LIN {X 0,Y 210.805,Z 412.053,A -85,B 0,C 180,E1 21926.273,E2 21926.273} C_VEL
LIN {X 0,Y 212.909,Z 406.81,A -85,B 0,C 180,E1 21927.449,E2 21927.449} C_VEL
LIN {X 0,Y 212.66,Z 395.692,A -85,B 0,C 180,E1 21932.561,E2 21932.561} C_VEL
LIN {X 0,Y 211.519,Z 388.072,A -85,B 0,C 180,E1 21938.035,E2 21938.035} C_VEL
LIN {X 0,Y 210.505,Z 384.471,A -85,B 0,C 180,E1 21943.363,E2 21943.363} C_VEL
LIN {X 0,Y 210.14,Z 383.897,A -85,B 0,C 180,E1 21947.585,E2 21947.585} C_VEL
LIN {X 0,Y 209.969,Z 386.924,A -85,B 0,C 180,E1 21953.986,E2 21953.986} C_VEL
LIN {X 0,Y 208.207,Z 395.855,A -85,B 0,C 180,E1 21960.026,E2 21960.026} C_VEL
LIN {X 0,Y 204.207,Z 408.112,A -85,B 0,C 180,E1 21965.858,E2 21965.858} C_VEL
LIN {X 0,Y 200.27,Z 414.736,A -85,B 0,C 180,E1 21968.169,E2 21968.169} C_VEL
LIN {X 0,Y 185.94,Z 431.439,A -85,B 0,C 180,E1 21974.122,E2 21974.122} C_VEL
LIN {X 0,Y 172.082,Z 443.956,A -85,B 0,C 180,E1 21982.208,E2 21982.208} C_VEL
LIN {X 0,Y 163.911,Z 449.524,A -85,B 0,C 180,E1 21989.305,E2 21989.305} C_VEL
LIN {X 0,Y 156.576,Z 451.973,A -85,B 0,C 180,E1 21999.559,E2 21999.559} C_VEL
LIN {X 0,Y 153.707,Z 449.459,A -85,B 0,C 180,E1 22009.428,E2 22009.428} C_VEL
LIN {X 0,Y 154.711,Z 442.064,A -85,B 0,C 180,E1 22019.51,E2 22019.51} C_VEL
LIN {X 0,Y 159.246,Z 429.175,A -85,B 0,C 180,E1 22029.201,E2 22029.201} C_VEL
LIN {X 0,Y 161.451,Z 424.273,A -85,B 0,C 180,E1 22032.224,E2 22032.224} C_VEL
LIN {X 0,Y 161.721,Z 426.86,A -85,B 0,C 180,E1 22033.746,E2 22033.746} C_VEL
LIN {X 0,Y 156.787,Z 439.27,A -85,B 0,C 180,E1 22041.701,E2 22041.701} C_VEL
LIN {X 0,Y 154.215,Z 446.583,A -85,B 0,C 180,E1 22050.002,E2 22050.002} C_VEL
LIN {X 0,Y 153.937,Z 447.484,A -85,B 0,C 180,E1 22051.727,E2 22051.727} C_VEL
LIN {X 0,Y 152.482,Z 449.035,A -85,B 0,C 180,E1 22054.89,E2 22054.89} C_VEL
LIN {X 0,Y 147.319,Z 450.78,A -85,B 0,C 180,E1 22063.882,E2 22063.882} C_VEL
LIN {X 0,Y 147.519,Z 450.447,A -85,B 0,C 180,E1 22064.726,E2 22064.726} C_VEL
LIN {X 0,Y 152.99,Z 446.068,A -85,B 0,C 180,E1 22074.785,E2 22074.785} C_VEL
LIN {X 0,Y 160.55,Z 436.902,A -85,B 0,C 180,E1 22083.051,E2 22083.051} C_VEL
LIN {X 0,Y 170.435,Z 421.674,A -85,B 0,C 180,E1 22090.476,E2 22090.476} C_VEL
LIN {X 0,Y 179.907,Z 402.515,A -85,B 0,C 180,E1 22095.907,E2 22095.907} C_VEL
LIN {X 0,Y 183.046,Z 393.253,A -85,B 0,C 180,E1 22097.899,E2 22097.899} C_VEL
LIN {X 0,Y 182.083,Z 375.139,A -85,B 0,C 180,E1 22103.032,E2 22103.032} C_VEL
LIN {X 0,Y 176.944,Z 356.373,A -85,B 0,C 180,E1 22108.755,E2 22108.755} C_VEL
LIN {X 0,Y 167.699,Z 337.888,A -85,B 0,C 180,E1 22116.078,E2 22116.078} C_VEL
LIN {X 0,Y 160.228,Z 325.849,A -85,B 0,C 180,E1 22123.781,E2 22123.781} C_VEL
LIN {X 0,Y 156.957,Z 319.955,A -85,B 0,C 180,E1 22128.879,E2 22128.879} C_VEL
LIN {X 0,Y 154.212,Z 314.241,A -85,B 0,C 180,E1 22136.459,E2 22136.459} C_VEL
LIN {X 0,Y 153.58,Z 313.235,A -85,B 0,C 180,E1 22142.781,E2 22142.781} C_VEL
LIN {X 0,Y 153.957,Z 314.585,A -85,B 0,C 180,E1 22147.024,E2 22147.024} C_VEL
LIN {X 0,Y 157.157,Z 320.346,A -85,B 0,C 180,E1 22155.852,E2 22155.852} C_VEL
LIN {X 0,Y 162.527,Z 330.048,A -85,B 0,C 180,E1 22163.386,E2 22163.386} C_VEL
LIN {X 0,Y 165.204,Z 338.961,A -85,B 0,C 180,E1 22166.589,E2 22166.589} C_VEL
LIN {X 0,Y 174.465,Z 373.972,A -85,B 0,C 180,E1 22175.303,E2 22175.303} C_VEL
LIN {X 0,Y 178.359,Z 393.841,A -85,B 0,C 180,E1 22179.484,E2 22179.484} C_VEL
LIN {X 0,Y 172.426,Z 418.787,A -85,B 0,C 180,E1 22182.402,E2 22182.402} C_VEL
LIN {X 0,Y 164.02,Z 441.927,A -85,B 0,C 180,E1 22187.123,E2 22187.123} C_VEL
LIN {X 0,Y 154.765,Z 462.181,A -85,B 0,C 180,E1 22194.194,E2 22194.194} C_VEL
LIN {X 0,Y 147.761,Z 476.495,A -85,B 0,C 180,E1 22202.64,E2 22202.64} C_VEL
LIN {X 0,Y 144.14,Z 485.452,A -85,B 0,C 180,E1 22211.694,E2 22211.694} C_VEL
LIN {X 0,Y 143.622,Z 488.993,A -85,B 0,C 180,E1 22217.868,E2 22217.868} C_VEL
LIN {X 0,Y 144.238,Z 490.637,A -85,B 0,C 180,E1 22223.993,E2 22223.993} C_VEL
LIN {X 0,Y 145.429,Z 490.426,A -85,B 0,C 180,E1 22229.998,E2 22229.998} C_VEL
LIN {X 0,Y 143.527,Z 490.304,A -85,B 0,C 180,E1 22242.137,E2 22242.137} C_VEL
LIN {X 0,Y 146.123,Z 485.431,A -85,B 0,C 180,E1 22254.396,E2 22254.396} C_VEL
LIN {X 0,Y 156.49,Z 474.216,A -85,B 0,C 180,E1 22267.06,E2 22267.06} C_VEL
LIN {X 0,Y 171.683,Z 458.424,A -85,B 0,C 180,E1 22276.477,E2 22276.477} C_VEL
LIN {X 0,Y 189.39,Z 437.637,A -85,B 0,C 180,E1 22283.408,E2 22283.408} C_VEL
LIN {X 0,Y 206.77,Z 412.673,A -85,B 0,C 180,E1 22288.125,E2 22288.125} C_VEL
LIN {X 0,Y 207.79,Z 406.319,A -85,B 0,C 180,E1 22290.626,E2 22290.626} C_VEL
LIN {X 0,Y 207.548,Z 396.618,A -85,B 0,C 180,E1 22296.457,E2 22296.457} C_VEL
LIN {X 0,Y 206.41,Z 391.41,A -85,B 0,C 180,E1 22303.023,E2 22303.023} C_VEL
LIN {X 0,Y 205.982,Z 390.645,A -85,B 0,C 180,E1 22307.331,E2 22307.331} C_VEL
LIN {X 0,Y 205.755,Z 391.801,A -85,B 0,C 180,E1 22311.592,E2 22311.592} C_VEL
LIN {X 0,Y 204.311,Z 397.423,A -85,B 0,C 180,E1 22316.851,E2 22316.851} C_VEL
LIN {X 0,Y 200.617,Z 407.807,A -85,B 0,C 180,E1 22322.722,E2 22322.722} C_VEL
LIN {X 0,Y 196.464,Z 415.576,A -85,B 0,C 180,E1 22326.12,E2 22326.12} C_VEL
LIN {X 0,Y 180.315,Z 433.31,A -85,B 0,C 180,E1 22332.5,E2 22332.5} C_VEL
LIN {X 0,Y 165.873,Z 445.381,A -85,B 0,C 180,E1 22340.582,E2 22340.582} C_VEL
LIN {X 0,Y 155.739,Z 451.419,A -85,B 0,C 180,E1 22349.308,E2 22349.308} C_VEL
LIN {X 0,Y 149.872,Z 453.121,A -85,B 0,C 180,E1 22357.212,E2 22357.212} C_VEL
LIN {X 0,Y 145.881,Z 450.344,A -85,B 0,C 180,E1 22369.442,E2 22369.442} C_VEL
LIN {X 0,Y 147.229,Z 441.856,A -85,B 0,C 180,E1 22380.841,E2 22380.841} C_VEL
LIN {X 0,Y 152.509,Z 427.688,A -85,B 0,C 180,E1 22391.256,E2 22391.256} C_VEL
LIN {X 0,Y 153.233,Z 427.258,A -85,B 0,C 180,E1 22392.085,E2 22392.085} C_VEL
LIN {X 0,Y 153.723,Z 429.514,A -85,B 0,C 180,E1 22393.609,E2 22393.609} C_VEL
LIN {X 0,Y 148.453,Z 442.037,A -85,B 0,C 180,E1 22402.702,E2 22402.702} C_VEL
LIN {X 0,Y 146.003,Z 449.201,A -85,B 0,C 180,E1 22412.964,E2 22412.964} C_VEL
LIN {X 0,Y 146.669,Z 450.944,A -85,B 0,C 180,E1 22421.876,E2 22421.876} C_VEL
LIN {X 0,Y 147.519,Z 450.447,A -85,B 0,C 180,E1 22424.726,E2 22424.726} C_VEL
LIN {X 0,Y 147.291,Z 449.557,A -85,B 0,C 180,E1 22429.824,E2 22429.824} C_VEL
LIN {X 0,Y 147.002,Z 445.958,A -85,B 0,C 180,E1 22437.425,E2 22437.425} C_VEL
LIN {X 0,Y 147.563,Z 445.28,A -85,B 0,C 180,E1 22438.211,E2 22438.211} C_VEL
LIN {X 0,Y 156.859,Z 433.988,A -85,B 0,C 180,E1 22446.962,E2 22446.962} C_VEL
LIN {X 0,Y 167.545,Z 417.022,A -85,B 0,C 180,E1 22454.121,E2 22454.121} C_VEL
LIN {X 0,Y 177.033,Z 396.635,A -85,B 0,C 180,E1 22459.12,E2 22459.12} C_VEL
LIN {X 0,Y 176.786,Z 379.155,A -85,B 0,C 180,E1 22464.405,E2 22464.405} C_VEL
LIN {X 0,Y 172.627,Z 361.262,A -85,B 0,C 180,E1 22470.275,E2 22470.275} C_VEL
LIN {X 0,Y 165.117,Z 344.486,A -85,B 0,C 180,E1 22477.286,E2 22477.286} C_VEL
LIN {X 0,Y 158.266,Z 332.872,A -85,B 0,C 180,E1 22484.958,E2 22484.958} C_VEL
LIN {X 0,Y 155.4,Z 327.402,A -85,B 0,C 180,E1 22489.872,E2 22489.872} C_VEL
LIN {X 0,Y 153.041,Z 321.347,A -85,B 0,C 180,E1 22497.669,E2 22497.669} C_VEL
LIN {X 0,Y 152.844,Z 322,A -85,B 0,C 180,E1 22506.075,E2 22506.075} C_VEL
LIN {X 0,Y 156.45,Z 329.767,A -85,B 0,C 180,E1 22516.569,E2 22516.569} C_VEL
LIN {X 0,Y 160.808,Z 337.775,A -85,B 0,C 180,E1 22522.738,E2 22522.738} C_VEL
LIN {X 0,Y 168.669,Z 370.735,A -85,B 0,C 180,E1 22531.861,E2 22531.861} C_VEL
LIN {X 0,Y 172.888,Z 396.716,A -85,B 0,C 180,E1 22537.69,E2 22537.69} C_VEL
LIN {X 0,Y 166.006,Z 421.766,A -85,B 0,C 180,E1 22540.92,E2 22540.92} C_VEL
LIN {X 0,Y 156.776,Z 444.406,A -85,B 0,C 180,E1 22546.023,E2 22546.023} C_VEL
LIN {X 0,Y 146.889,Z 463.923,A -85,B 0,C 180,E1 22553.634,E2 22553.634} C_VEL
LIN {X 0,Y 139.622,Z 477.386,A -85,B 0,C 180,E1 22562.654,E2 22562.654} C_VEL
LIN {X 0,Y 135.933,Z 486.411,A -85,B 0,C 180,E1 22573.886,E2 22573.886} C_VEL
LIN {X 0,Y 136.423,Z 489.615,A -85,B 0,C 180,E1 22584.182,E2 22584.182} C_VEL
LIN {X 0,Y 137.542,Z 489.303,A -85,B 0,C 180,E1 22589.998,E2 22589.998} C_VEL
LIN {X 0,Y 135.654,Z 489.171,A -85,B 0,C 180,E1 22602.853,E2 22602.853} C_VEL
LIN {X 0,Y 138.762,Z 484.534,A -85,B 0,C 180,E1 22615.782,E2 22615.782} C_VEL
LIN {X 0,Y 150.121,Z 473.656,A -85,B 0,C 180,E1 22628.918,E2 22628.918} C_VEL
LIN {X 0,Y 167.438,Z 457.052,A -85,B 0,C 180,E1 22639.004,E2 22639.004} C_VEL
LIN {X 0,Y 186.696,Z 435.597,A -85,B 0,C 180,E1 22645.939,E2 22645.939} C_VEL
LIN {X 0,Y 202.13,Z 414.122,A -85,B 0,C 180,E1 22650.063,E2 22650.063} C_VEL
LIN {X 0,Y 202.743,Z 404.443,A -85,B 0,C 180,E1 22655.64,E2 22655.64} C_VEL
LIN {X 0,Y 202.276,Z 398.832,A -85,B 0,C 180,E1 22661.292,E2 22661.292} C_VEL
LIN {X 0,Y 201.541,Z 397.217,A -85,B 0,C 180,E1 22667.047,E2 22667.047} C_VEL
LIN {X 0,Y 201.127,Z 398.232,A -85,B 0,C 180,E1 22671.397,E2 22671.397} C_VEL
LIN {X 0,Y 198.994,Z 403.913,A -85,B 0,C 180,E1 22676.767,E2 22676.767} C_VEL
LIN {X 0,Y 194.16,Z 414.133,A -85,B 0,C 180,E1 22682.645,E2 22682.645} C_VEL
LIN {X 0,Y 190.211,Z 419.697,A -85,B 0,C 180,E1 22684.884,E2 22684.884} C_VEL
LIN {X 0,Y 172.815,Z 436.956,A -85,B 0,C 180,E1 22691.686,E2 22691.686} C_VEL
LIN {X 0,Y 159.581,Z 446.936,A -85,B 0,C 180,E1 22698.991,E2 22698.991} C_VEL
LIN {X 0,Y 150.897,Z 451.871,A -85,B 0,C 180,E1 22705.844,E2 22705.844} C_VEL
LIN {X 0,Y 144.368,Z 454.101,A -85,B 0,C 180,E1 22713.263,E2 22713.263} C_VEL
LIN {X 0,Y 139.14,Z 453.339,A -85,B 0,C 180,E1 22723.652,E2 22723.652} C_VEL
LIN {X 0,Y 138.099,Z 447.736,A -85,B 0,C 180,E1 22735.228,E2 22735.228} C_VEL
LIN {X 0,Y 141.88,Z 436.027,A -85,B 0,C 180,E1 22747.02,E2 22747.02} C_VEL
LIN {X 0,Y 144.913,Z 429.972,A -85,B 0,C 180,E1 22751.798,E2 22751.798} C_VEL
LIN {X 0,Y 146.25,Z 430.872,A -85,B 0,C 180,E1 22752.746,E2 22752.746} C_VEL
LIN {X 0,Y 140.701,Z 443.288,A -85,B 0,C 180,E1 22762.297,E2 22762.297} C_VEL
LIN {X 0,Y 138.16,Z 450.352,A -85,B 0,C 180,E1 22773.132,E2 22773.132} C_VEL
LIN {X 0,Y 139.006,Z 452.016,A -85,B 0,C 180,E1 22782.541,E2 22782.541} C_VEL
LIN {X 0,Y 142.983,Z 449.701,A -85,B 0,C 180,E1 22791.679,E2 22791.679} C_VEL
LIN {X 0,Y 147.563,Z 445.28,A -85,B 0,C 180,E1 22798.211,E2 22798.211} C_VEL
LIN {X 0,Y 149.721,Z 439.575,A -85,B 0,C 180,E1 22804.559,E2 22804.559} C_VEL
LIN {X 0,Y 152.089,Z 432.976,A -85,B 0,C 180,E1 22809.758,E2 22809.758} C_VEL
LIN {X 0,Y 152.872,Z 431.795,A -85,B 0,C 180,E1 22810.388,E2 22810.388} C_VEL
LIN {X 0,Y 163.705,Z 414.626,A -85,B 0,C 180,E1 22816.989,E2 22816.989} C_VEL
LIN {X 0,Y 171.296,Z 398.113,A -85,B 0,C 180,E1 22821.011,E2 22821.011} C_VEL
LIN {X 0,Y 171.365,Z 380.746,A -85,B 0,C 180,E1 22826.61,E2 22826.61} C_VEL
LIN {X 0,Y 167.41,Z 363.025,A -85,B 0,C 180,E1 22833.065,E2 22833.065} C_VEL
LIN {X 0,Y 160.467,Z 346.936,A -85,B 0,C 180,E1 22840.83,E2 22840.83} C_VEL
LIN {X 0,Y 154.104,Z 335.035,A -85,B 0,C 180,E1 22850.453,E2 22850.453} C_VEL
LIN {X 0,Y 151.767,Z 328.746,A -85,B 0,C 180,E1 22859.964,E2 22859.964} C_VEL
LIN {X 0,Y 151.796,Z 329.901,A -85,B 0,C 180,E1 22865.67,E2 22865.67} C_VEL
LIN {X 0,Y 154.905,Z 337.215,A -85,B 0,C 180,E1 22875.684,E2 22875.684} C_VEL
LIN {X 0,Y 158.461,Z 344.268,A -85,B 0,C 180,E1 22881.252,E2 22881.252} C_VEL
LIN {X 0,Y 165.451,Z 378.334,A -85,B 0,C 180,E1 22890.84,E2 22890.84} C_VEL
LIN {X 0,Y 167.53,Z 399.638,A -85,B 0,C 180,E1 22895.837,E2 22895.837} C_VEL
LIN {X 0,Y 159.333,Z 425.462,A -85,B 0,C 180,E1 22899.527,E2 22899.527} C_VEL
LIN {X 0,Y 148.853,Z 448.162,A -85,B 0,C 180,E1 22905.324,E2 22905.324} C_VEL
LIN {X 0,Y 138.78,Z 465.913,A -85,B 0,C 180,E1 22913.269,E2 22913.269} C_VEL
LIN {X 0,Y 131.489,Z 478.074,A -85,B 0,C 180,E1 22922.672,E2 22922.672} C_VEL
LIN {X 0,Y 128.162,Z 485.373,A -85,B 0,C 180,E1 22932.879,E2 22932.879} C_VEL
LIN {X 0,Y 128.366,Z 488.45,A -85,B 0,C 180,E1 22943.247,E2 22943.247} C_VEL
LIN {X 0,Y 129.676,Z 488.176,A -85,B 0,C 180,E1 22949.998,E2 22949.998} C_VEL
LIN {X 0,Y 127.83,Z 488.043,A -85,B 0,C 180,E1 22963.654,E2 22963.654} C_VEL
LIN {X 0,Y 131.494,Z 483.615,A -85,B 0,C 180,E1 22977.323,E2 22977.323} C_VEL
LIN {X 0,Y 143.906,Z 473.073,A -85,B 0,C 180,E1 22990.946,E2 22990.946} C_VEL
LIN {X 0,Y 162.302,Z 456.894,A -85,B 0,C 180,E1 23001.136,E2 23001.136} C_VEL
LIN {X 0,Y 180.943,Z 437.582,A -85,B 0,C 180,E1 23007.604,E2 23007.604} C_VEL
LIN {X 0,Y 196.06,Z 418.633,A -85,B 0,C 180,E1 23011.375,E2 23011.375} C_VEL
LIN {X 0,Y 197.333,Z 413.38,A -85,B 0,C 180,E1 23013.946,E2 23013.946} C_VEL
LIN {X 0,Y 197.677,Z 406.978,A -85,B 0,C 180,E1 23019.037,E2 23019.037} C_VEL
LIN {X 0,Y 197.396,Z 404.738,A -85,B 0,C 180,E1 23022.223,E2 23022.223} C_VEL
LIN {X 0,Y 196.826,Z 403.614,A -85,B 0,C 180,E1 23026.731,E2 23026.731} C_VEL
LIN {X 0,Y 196.239,Z 404.454,A -85,B 0,C 180,E1 23031.181,E2 23031.181} C_VEL
LIN {X 0,Y 194.096,Z 408.723,A -85,B 0,C 180,E1 23035.569,E2 23035.569} C_VEL
LIN {X 0,Y 188.715,Z 418.042,A -85,B 0,C 180,E1 23041.394,E2 23041.394} C_VEL
LIN {X 0,Y 184.124,Z 423.609,A -85,B 0,C 180,E1 23043.541,E2 23043.541} C_VEL
LIN {X 0,Y 168.281,Z 438.119,A -85,B 0,C 180,E1 23049.475,E2 23049.475} C_VEL
LIN {X 0,Y 153.567,Z 448.438,A -85,B 0,C 180,E1 23057.182,E2 23057.182} C_VEL
LIN {X 0,Y 143.496,Z 453.5,A -85,B 0,C 180,E1 23064.917,E2 23064.917} C_VEL
LIN {X 0,Y 133.608,Z 455.364,A -85,B 0,C 180,E1 23077.762,E2 23077.762} C_VEL
LIN {X 0,Y 130.093,Z 451.283,A -85,B 0,C 180,E1 23090.894,E2 23090.894} C_VEL
LIN {X 0,Y 132.032,Z 442.347,A -85,B 0,C 180,E1 23102.798,E2 23102.798} C_VEL
LIN {X 0,Y 136.522,Z 432.65,A -85,B 0,C 180,E1 23111.473,E2 23111.473} C_VEL
LIN {X 0,Y 138.032,Z 433.439,A -85,B 0,C 180,E1 23112.506,E2 23112.506} C_VEL
LIN {X 0,Y 132.977,Z 444.536,A -85,B 0,C 180,E1 23121.847,E2 23121.847} C_VEL
LIN {X 0,Y 130.321,Z 451.504,A -85,B 0,C 180,E1 23133.321,E2 23133.321} C_VEL
LIN {X 0,Y 131.334,Z 453.091,A -85,B 0,C 180,E1 23143.287,E2 23143.287} C_VEL
LIN {X 0,Y 135.672,Z 450.7,A -85,B 0,C 180,E1 23152.912,E2 23152.912} C_VEL
LIN {X 0,Y 143.946,Z 442.74,A -85,B 0,C 180,E1 23163.212,E2 23163.212} C_VEL
LIN {X 0,Y 152.872,Z 431.795,A -85,B 0,C 180,E1 23170.388,E2 23170.388} C_VEL
LIN {X 0,Y 156.693,Z 422.244,A -85,B 0,C 180,E1 23175.64,E2 23175.64} C_VEL
LIN {X 0,Y 159.956,Z 412.576,A -85,B 0,C 180,E1 23179.794,E2 23179.794} C_VEL
LIN {X 0,Y 160.772,Z 410.96,A -85,B 0,C 180,E1 23180.247,E2 23180.247} C_VEL
LIN {X 0,Y 165.708,Z 399.848,A -85,B 0,C 180,E1 23182.948,E2 23182.948} C_VEL
LIN {X 0,Y 166.113,Z 382.865,A -85,B 0,C 180,E1 23188.852,E2 23188.852} C_VEL
LIN {X 0,Y 162.778,Z 365.829,A -85,B 0,C 180,E1 23195.684,E2 23195.684} C_VEL
LIN {X 0,Y 157.291,Z 352.144,A -85,B 0,C 180,E1 23203.237,E2 23203.237} C_VEL
LIN {X 0,Y 152.493,Z 342.283,A -85,B 0,C 180,E1 23211.789,E2 23211.789} C_VEL
LIN {X 0,Y 150.797,Z 336.592,A -85,B 0,C 180,E1 23219.964,E2 23219.964} C_VEL
LIN {X 0,Y 150.78,Z 337.933,A -85,B 0,C 180,E1 23225.528,E2 23225.528} C_VEL
LIN {X 0,Y 153.465,Z 344.797,A -85,B 0,C 180,E1 23234.922,E2 23234.922} C_VEL
LIN {X 0,Y 156.314,Z 351.22,A -85,B 0,C 180,E1 23239.895,E2 23239.895} C_VEL
LIN {X 0,Y 161.485,Z 382.794,A -85,B 0,C 180,E1 23249.038,E2 23249.038} C_VEL
LIN {X 0,Y 162.32,Z 402.187,A -85,B 0,C 180,E1 23253.864,E2 23253.864} C_VEL
LIN {X 0,Y 153.779,Z 426.313,A -85,B 0,C 180,E1 23257.493,E2 23257.493} C_VEL
LIN {X 0,Y 142.508,Z 448.71,A -85,B 0,C 180,E1 23263.494,E2 23263.494} C_VEL
LIN {X 0,Y 131.555,Z 466.294,A -85,B 0,C 180,E1 23271.934,E2 23271.934} C_VEL
LIN {X 0,Y 123.393,Z 478.609,A -85,B 0,C 180,E1 23282.701,E2 23282.701} C_VEL
LIN {X 0,Y 120.059,Z 485.795,A -85,B 0,C 180,E1 23295.439,E2 23295.439} C_VEL
LIN {X 0,Y 120.873,Z 487.433,A -85,B 0,C 180,E1 23306.366,E2 23306.366} C_VEL
LIN {X 0,Y 121.317,Z 486.688,A -85,B 0,C 180,E1 23311.908,E2 23311.908} C_VEL
LIN {X 0,Y 120.005,Z 486.912,A -85,B 0,C 180,E1 23324.563,E2 23324.563} C_VEL
LIN {X 0,Y 126.284,Z 481.233,A -85,B 0,C 180,E1 23341.962,E2 23341.962} C_VEL
LIN {X 0,Y 139.924,Z 471.028,A -85,B 0,C 180,E1 23354.504,E2 23354.504} C_VEL
LIN {X 0,Y 160.011,Z 454.469,A -85,B 0,C 180,E1 23364.426,E2 23364.426} C_VEL
LIN {X 0,Y 179.816,Z 434.786,A -85,B 0,C 180,E1 23370.532,E2 23370.532} C_VEL
LIN {X 0,Y 191.147,Z 421.174,A -85,B 0,C 180,E1 23373.152,E2 23373.152} C_VEL
LIN {X 0,Y 192.528,Z 413.608,A -85,B 0,C 180,E1 23378.568,E2 23378.568} C_VEL
LIN {X 0,Y 192.418,Z 411.209,A -85,B 0,C 180,E1 23381.747,E2 23381.747} C_VEL
LIN {X 0,Y 191.854,Z 409.833,A -85,B 0,C 180,E1 23386.38,E2 23386.38} C_VEL
LIN {X 0,Y 191.109,Z 410.493,A -85,B 0,C 180,E1 23390.942,E2 23390.942} C_VEL
LIN {X 0,Y 188.294,Z 414.857,A -85,B 0,C 180,E1 23395.432,E2 23395.432} C_VEL
LIN {X 0,Y 182.741,Z 422.708,A -85,B 0,C 180,E1 23400.502,E2 23400.502} C_VEL
LIN {X 0,Y 164.382,Z 439.097,A -85,B 0,C 180,E1 23406.999,E2 23406.999} C_VEL
LIN {X 0,Y 146.552,Z 450.584,A -85,B 0,C 180,E1 23415.965,E2 23415.965} C_VEL
LIN {X 0,Y 133.074,Z 456.024,A -85,B 0,C 180,E1 23427.02,E2 23427.02} C_VEL
LIN {X 0,Y 126.093,Z 456.508,A -85,B 0,C 180,E1 23436.808,E2 23436.808} C_VEL
LIN {X 0,Y 122.301,Z 452.626,A -85,B 0,C 180,E1 23449.795,E2 23449.795} C_VEL
LIN {X 0,Y 124.386,Z 442.778,A -85,B 0,C 180,E1 23463.664,E2 23463.664} C_VEL
LIN {X 0,Y 127.906,Z 435.011,A -85,B 0,C 180,E1 23470.835,E2 23470.835} C_VEL
LIN {X 0,Y 129.937,Z 436.257,A -85,B 0,C 180,E1 23472.517,E2 23472.517} C_VEL
LIN {X 0,Y 124.598,Z 447.108,A -85,B 0,C 180,E1 23483.046,E2 23483.046} C_VEL
LIN {X 0,Y 122.496,Z 452.653,A -85,B 0,C 180,E1 23493.533,E2 23493.533} C_VEL
LIN {X 0,Y 123.686,Z 454.166,A -85,B 0,C 180,E1 23504.125,E2 23504.125} C_VEL
LIN {X 0,Y 128.447,Z 451.697,A -85,B 0,C 180,E1 23514.281,E2 23514.281} C_VEL
LIN {X 0,Y 137.57,Z 443.46,A -85,B 0,C 180,E1 23525.163,E2 23525.163} C_VEL
LIN {X 0,Y 148.385,Z 430.671,A -85,B 0,C 180,E1 23533.351,E2 23533.351} C_VEL
LIN {X 0,Y 159.898,Z 412.582,A -85,B 0,C 180,E1 23539.819,E2 23539.819} C_VEL
LIN {X 0,Y 160.772,Z 410.96,A -85,B 0,C 180,E1 23540.247,E2 23540.247} C_VEL
LIN {X 0,Y 162.059,Z 405.175,A -85,B 0,C 180,E1 23542.492,E2 23542.492} C_VEL
LIN {X 0,Y 160.978,Z 396.411,A -85,B 0,C 180,E1 23546.913,E2 23546.913} C_VEL
LIN {X 0,Y 160.558,Z 379.637,A -85,B 0,C 180,E1 23553.447,E2 23553.447} C_VEL
LIN {X 0,Y 156.861,Z 363.892,A -85,B 0,C 180,E1 23561.199,E2 23561.199} C_VEL
LIN {X 0,Y 152.459,Z 353.028,A -85,B 0,C 180,E1 23569.366,E2 23569.366} C_VEL
LIN {X 0,Y 150.687,Z 349.088,A -85,B 0,C 180,E1 23573.988,E2 23573.988} C_VEL
LIN {X 0,Y 149.83,Z 344.417,A -85,B 0,C 180,E1 23579.964,E2 23579.964} C_VEL
LIN {X 0,Y 149.754,Z 345.853,A -85,B 0,C 180,E1 23585.203,E2 23585.203} C_VEL
LIN {X 0,Y 152.127,Z 352.59,A -85,B 0,C 180,E1 23594.322,E2 23594.322} C_VEL
LIN {X 0,Y 154.171,Z 357.768,A -85,B 0,C 180,E1 23598.327,E2 23598.327} C_VEL
LIN {X 0,Y 157.398,Z 386.382,A -85,B 0,C 180,E1 23606.92,E2 23606.92} C_VEL
LIN {X 0,Y 157.312,Z 404.479,A -85,B 0,C 180,E1 23611.75,E2 23611.75} C_VEL
LIN {X 0,Y 147.518,Z 429.048,A -85,B 0,C 180,E1 23615.711,E2 23615.711} C_VEL
LIN {X 0,Y 135.243,Z 450.893,A -85,B 0,C 180,E1 23622.148,E2 23622.148} C_VEL
LIN {X 0,Y 123.57,Z 467.694,A -85,B 0,C 180,E1 23631.253,E2 23631.253} C_VEL
LIN {X 0,Y 115.288,Z 479.002,A -85,B 0,C 180,E1 23642.732,E2 23642.732} C_VEL
LIN {X 0,Y 112.271,Z 484.727,A -85,B 0,C 180,E1 23654.404,E2 23654.404} C_VEL
LIN {X 0,Y 112.491,Z 486.26,A -85,B 0,C 180,E1 23662.289,E2 23662.289} C_VEL
LIN {X 0,Y 113.889,Z 485.895,A -85,B 0,C 180,E1 23669.998,E2 23669.998} C_VEL
LIN {X 0,Y 112.238,Z 485.719,A -85,B 0,C 180,E1 23685.596,E2 23685.596} C_VEL
LIN {X 0,Y 119.281,Z 480.544,A -85,B 0,C 180,E1 23703.777,E2 23703.777} C_VEL
LIN {X 0,Y 135.655,Z 469.585,A -85,B 0,C 180,E1 23717.764,E2 23717.764} C_VEL
LIN {X 0,Y 156.889,Z 453.28,A -85,B 0,C 180,E1 23727.306,E2 23727.306} C_VEL
LIN {X 0,Y 179.167,Z 431.933,A -85,B 0,C 180,E1 23733.489,E2 23733.489} C_VEL
LIN {X 0,Y 185.462,Z 424.819,A -85,B 0,C 180,E1 23734.819,E2 23734.819} C_VEL
LIN {X 0,Y 186.889,Z 420.362,A -85,B 0,C 180,E1 23737.888,E2 23737.888} C_VEL
LIN {X 0,Y 187.131,Z 417.51,A -85,B 0,C 180,E1 23741.212,E2 23741.212} C_VEL
LIN {X 0,Y 186.605,Z 415.856,A -85,B 0,C 180,E1 23746.017,E2 23746.017} C_VEL
LIN {X 0,Y 185.698,Z 416.347,A -85,B 0,C 180,E1 23750.676,E2 23750.676} C_VEL
LIN {X 0,Y 181.541,Z 421.568,A -85,B 0,C 180,E1 23755.892,E2 23755.892} C_VEL
LIN {X 0,Y 177.832,Z 425.976,A -85,B 0,C 180,E1 23758.814,E2 23758.814} C_VEL
LIN {X 0,Y 157.972,Z 442.127,A -85,B 0,C 180,E1 23765.516,E2 23765.516} C_VEL
LIN {X 0,Y 140.138,Z 452.46,A -85,B 0,C 180,E1 23774.284,E2 23774.284} C_VEL
LIN {X 0,Y 129.968,Z 456.39,A -85,B 0,C 180,E1 23781.75,E2 23781.75} C_VEL
LIN {X 0,Y 122.156,Z 457.854,A -85,B 0,C 180,E1 23790.154,E2 23790.154} C_VEL
LIN {X 0,Y 115.289,Z 455.59,A -85,B 0,C 180,E1 23804.342,E2 23804.342} C_VEL
LIN {X 0,Y 114.969,Z 448.327,A -85,B 0,C 180,E1 23818.334,E2 23818.334} C_VEL
LIN {X 0,Y 119.593,Z 437.622,A -85,B 0,C 180,E1 23830.482,E2 23830.482} C_VEL
LIN {X 0,Y 121.648,Z 439.376,A -85,B 0,C 180,E1 23832.902,E2 23832.902} C_VEL
LIN {X 0,Y 116.258,Z 449.535,A -85,B 0,C 180,E1 23844.416,E2 23844.416} C_VEL
LIN {X 0,Y 114.654,Z 454.745,A -85,B 0,C 180,E1 23857.565,E2 23857.565} C_VEL
LIN {X 0,Y 116.069,Z 455.241,A -85,B 0,C 180,E1 23865.073,E2 23865.073} C_VEL
LIN {X 0,Y 121.287,Z 452.698,A -85,B 0,C 180,E1 23875.816,E2 23875.816} C_VEL
LIN {X 0,Y 131.184,Z 444.352,A -85,B 0,C 180,E1 23887.152,E2 23887.152} C_VEL
LIN {X 0,Y 142.732,Z 431.433,A -85,B 0,C 180,E1 23895.533,E2 23895.533} C_VEL
LIN {X 0,Y 154.947,Z 413.14,A -85,B 0,C 180,E1 23902.064,E2 23902.064} C_VEL
LIN {X 0,Y 160.269,Z 401.818,A -85,B 0,C 180,E1 23904.94,E2 23904.94} C_VEL
LIN {X 0,Y 160.978,Z 396.411,A -85,B 0,C 180,E1 23906.913,E2 23906.913} C_VEL
LIN {X 0,Y 159.626,Z 389.093,A -85,B 0,C 180,E1 23910.776,E2 23910.776} C_VEL
LIN {X 0,Y 155.49,Z 378.673,A -85,B 0,C 180,E1 23917.838,E2 23917.838} C_VEL
LIN {X 0,Y 152.589,Z 365.981,A -85,B 0,C 180,E1 23925.466,E2 23925.466} C_VEL
LIN {X 0,Y 149.683,Z 357.153,A -85,B 0,C 180,E1 23933.815,E2 23933.815} C_VEL
LIN {X 0,Y 148.755,Z 352.334,A -85,B 0,C 180,E1 23941.417,E2 23941.417} C_VEL
LIN {X 0,Y 148.808,Z 355.001,A -85,B 0,C 180,E1 23946.332,E2 23946.332} C_VEL
LIN {X 0,Y 150.809,Z 360.325,A -85,B 0,C 180,E1 23953.711,E2 23953.711} C_VEL
LIN {X 0,Y 152.128,Z 364.314,A -85,B 0,C 180,E1 23956.718,E2 23956.718} C_VEL
LIN {X 0,Y 153.43,Z 390.946,A -85,B 0,C 180,E1 23965.06,E2 23965.06} C_VEL
LIN {X 0,Y 152.653,Z 406.086,A -85,B 0,C 180,E1 23969.424,E2 23969.424} C_VEL
LIN {X 0,Y 142.319,Z 429.75,A -85,B 0,C 180,E1 23973.383,E2 23973.383} C_VEL
LIN {X 0,Y 129.981,Z 450.139,A -85,B 0,C 180,E1 23979.518,E2 23979.518} C_VEL
LIN {X 0,Y 117.353,Z 466.806,A -85,B 0,C 180,E1 23988.773,E2 23988.773} C_VEL
LIN {X 0,Y 108.126,Z 478.001,A -85,B 0,C 180,E1 24000.758,E2 24000.758} C_VEL
LIN {X 0,Y 104.507,Z 483.656,A -85,B 0,C 180,E1 24013.212,E2 24013.212} C_VEL
LIN {X 0,Y 104.554,Z 485.162,A -85,B 0,C 180,E1 24021.699,E2 24021.699} C_VEL
LIN {X 0,Y 105.974,Z 484.758,A -85,B 0,C 180,E1 24029.998,E2 24029.998} C_VEL
LIN {X 0,Y 104.5,Z 484.512,A -85,B 0,C 180,E1 24046.784,E2 24046.784} C_VEL
LIN {X 0,Y 110.446,Z 480.927,A -85,B 0,C 180,E1 24063.125,E2 24063.125} C_VEL
LIN {X 0,Y 126.155,Z 471.758,A -85,B 0,C 180,E1 24077.855,E2 24077.855} C_VEL
LIN {X 0,Y 148.416,Z 456.636,A -85,B 0,C 180,E1 24088.374,E2 24088.374} C_VEL
LIN {X 0,Y 171.01,Z 437.373,A -85,B 0,C 180,E1 24094.748,E2 24094.748} C_VEL
LIN {X 0,Y 180.634,Z 427.453,A -85,B 0,C 180,E1 24096.766,E2 24096.766} C_VEL
LIN {X 0,Y 181.503,Z 423.664,A -85,B 0,C 180,E1 24100.607,E2 24100.607} C_VEL
LIN {X 0,Y 181.089,Z 421.688,A -85,B 0,C 180,E1 24105.554,E2 24105.554} C_VEL
LIN {X 0,Y 180.038,Z 421.976,A -85,B 0,C 180,E1 24110.38,E2 24110.38} C_VEL
LIN {X 0,Y 175.68,Z 426.509,A -85,B 0,C 180,E1 24115.103,E2 24115.103} C_VEL
LIN {X 0,Y 171.277,Z 430.697,A -85,B 0,C 180,E1 24117.538,E2 24117.538} C_VEL
LIN {X 0,Y 151.274,Z 445.268,A -85,B 0,C 180,E1 24124.057,E2 24124.057} C_VEL
LIN {X 0,Y 132.623,Z 454.754,A -85,B 0,C 180,E1 24133.196,E2 24133.196} C_VEL
LIN {X 0,Y 117.336,Z 458.941,A -85,B 0,C 180,E1 24145.816,E2 24145.816} C_VEL
LIN {X 0,Y 108.422,Z 457.454,A -85,B 0,C 180,E1 24160.729,E2 24160.729} C_VEL
LIN {X 0,Y 106.689,Z 451.076,A -85,B 0,C 180,E1 24175.548,E2 24175.548} C_VEL
LIN {X 0,Y 110.946,Z 439.866,A -85,B 0,C 180,E1 24189.622,E2 24189.622} C_VEL
LIN {X 0,Y 113.531,Z 441.851,A -85,B 0,C 180,E1 24192.838,E2 24192.838} C_VEL
LIN {X 0,Y 107.926,Z 451.831,A -85,B 0,C 180,E1 24205.994,E2 24205.994} C_VEL
LIN {X 0,Y 106.91,Z 455.914,A -85,B 0,C 180,E1 24218.529,E2 24218.529} C_VEL
LIN {X 0,Y 108.488,Z 456.317,A -85,B 0,C 180,E1 24226.154,E2 24226.154} C_VEL
LIN {X 0,Y 114.235,Z 453.697,A -85,B 0,C 180,E1 24237.54,E2 24237.54} C_VEL
LIN {X 0,Y 124.973,Z 445.243,A -85,B 0,C 180,E1 24249.342,E2 24249.342} C_VEL
LIN {X 0,Y 137.307,Z 432.189,A -85,B 0,C 180,E1 24257.889,E2 24257.889} C_VEL
LIN {X 0,Y 149.974,Z 414.138,A -85,B 0,C 180,E1 24264.332,E2 24264.332} C_VEL
LIN {X 0,Y 154.856,Z 404.456,A -85,B 0,C 180,E1 24266.85,E2 24266.85} C_VEL
LIN {X 0,Y 156.332,Z 387.632,A -85,B 0,C 180,E1 24273.645,E2 24273.645} C_VEL
LIN {X 0,Y 155.49,Z 378.673,A -85,B 0,C 180,E1 24277.838,E2 24277.838} C_VEL
LIN {X 0,Y 153.28,Z 373.334,A -85,B 0,C 180,E1 24282.195,E2 24282.195} C_VEL
LIN {X 0,Y 148.904,Z 368.422,A -85,B 0,C 180,E1 24290.376,E2 24290.376} C_VEL
LIN {X 0,Y 147.817,Z 363.771,A -85,B 0,C 180,E1 24296.122,E2 24296.122} C_VEL
LIN {X 0,Y 147.713,Z 360.172,A -85,B 0,C 180,E1 24302.159,E2 24302.159} C_VEL
LIN {X 0,Y 149.322,Z 368.019,A -85,B 0,C 180,E1 24313.106,E2 24313.106} C_VEL
LIN {X 0,Y 149.907,Z 371.434,A -85,B 0,C 180,E1 24315.285,E2 24315.285} C_VEL
LIN {X 0,Y 149.22,Z 397.655,A -85,B 0,C 180,E1 24323.821,E2 24323.821} C_VEL
LIN {X 0,Y 147.791,Z 408.695,A -85,B 0,C 180,E1 24327.098,E2 24327.098} C_VEL
LIN {X 0,Y 135.938,Z 432.823,A -85,B 0,C 180,E1 24331.418,E2 24331.418} C_VEL
LIN {X 0,Y 122.131,Z 453.125,A -85,B 0,C 180,E1 24338.283,E2 24338.283} C_VEL
LIN {X 0,Y 108.675,Z 468.88,A -85,B 0,C 180,E1 24348.554,E2 24348.554} C_VEL
LIN {X 0,Y 99.068,Z 479.331,A -85,B 0,C 180,E1 24362.806,E2 24362.806} C_VEL
LIN {X 0,Y 96.793,Z 482.585,A -85,B 0,C 180,E1 24371.83,E2 24371.83} C_VEL
LIN {X 0,Y 96.629,Z 484.06,A -85,B 0,C 180,E1 24381.013,E2 24381.013} C_VEL
LIN {X 0,Y 98.086,Z 483.626,A -85,B 0,C 180,E1 24389.997,E2 24389.997} C_VEL
LIN {X 0,Y 97.289,Z 482.811,A -85,B 0,C 180,E1 24394.445,E2 24394.445} C_VEL
LIN {X 0,Y 97.472,Z 483.009,A -85,B 0,C 180,E1 24411.883,E2 24411.883} C_VEL
LIN {X 0,Y 107.182,Z 478.298,A -85,B 0,C 180,E1 24429.817,E2 24429.817} C_VEL
LIN {X 0,Y 126.214,Z 468.153,A -85,B 0,C 180,E1 24443.678,E2 24443.678} C_VEL
LIN {X 0,Y 150.389,Z 452.198,A -85,B 0,C 180,E1 24452.934,E2 24452.934} C_VEL
LIN {X 0,Y 174.5,Z 431.507,A -85,B 0,C 180,E1 24458.498,E2 24458.498} C_VEL
LIN {X 0,Y 175.645,Z 428.923,A -85,B 0,C 180,E1 24460.909,E2 24460.909} C_VEL
LIN {X 0,Y 175.3,Z 427.308,A -85,B 0,C 180,E1 24465.066,E2 24465.066} C_VEL
LIN {X 0,Y 174.116,Z 427.389,A -85,B 0,C 180,E1 24470.05,E2 24470.05} C_VEL
LIN {X 0,Y 170.441,Z 430.59,A -85,B 0,C 180,E1 24473.678,E2 24473.678} C_VEL
LIN {X 0,Y 166.475,Z 433.94,A -85,B 0,C 180,E1 24475.604,E2 24475.604} C_VEL
LIN {X 0,Y 145.99,Z 447.605,A -85,B 0,C 180,E1 24481.957,E2 24481.957} C_VEL
LIN {X 0,Y 127.154,Z 456.273,A -85,B 0,C 180,E1 24490.761,E2 24490.761} C_VEL
LIN {X 0,Y 110.128,Z 460.237,A -85,B 0,C 180,E1 24504.326,E2 24504.326} C_VEL
LIN {X 0,Y 100.302,Z 457.987,A -85,B 0,C 180,E1 24521.22,E2 24521.22} C_VEL
LIN {X 0,Y 99.341,Z 449.683,A -85,B 0,C 180,E1 24539.228,E2 24539.228} C_VEL
LIN {X 0,Y 102.48,Z 442.264,A -85,B 0,C 180,E1 24548.94,E2 24548.94} C_VEL
LIN {X 0,Y 105.026,Z 444.798,A -85,B 0,C 180,E1 24553.303,E2 24553.303} C_VEL
LIN {X 0,Y 100.119,Z 453.017,A -85,B 0,C 180,E1 24565.681,E2 24565.681} C_VEL
LIN {X 0,Y 99.099,Z 456.97,A -85,B 0,C 180,E1 24578.761,E2 24578.761} C_VEL
LIN {X 0,Y 100.951,Z 457.393,A -85,B 0,C 180,E1 24587.397,E2 24587.397} C_VEL
LIN {X 0,Y 107.291,Z 454.697,A -85,B 0,C 180,E1 24599.492,E2 24599.492} C_VEL
LIN {X 0,Y 118.979,Z 446.132,A -85,B 0,C 180,E1 24611.75,E2 24611.75} C_VEL
LIN {X 0,Y 132.13,Z 432.947,A -85,B 0,C 180,E1 24620.437,E2 24620.437} C_VEL
LIN {X 0,Y 145.776,Z 414.244,A -85,B 0,C 180,E1 24626.995,E2 24626.995} C_VEL
LIN {X 0,Y 149.707,Z 406.674,A -85,B 0,C 180,E1 24629.052,E2 24629.052} C_VEL
LIN {X 0,Y 151.711,Z 391.308,A -85,B 0,C 180,E1 24635.737,E2 24635.737} C_VEL
LIN {X 0,Y 150.756,Z 377.471,A -85,B 0,C 180,E1 24643.237,E2 24643.237} C_VEL
LIN {X 0,Y 148.904,Z 368.422,A -85,B 0,C 180,E1 24650.376,E2 24650.376} C_VEL
LIN {X 0,Y 147.558,Z 368.261,A -85,B 0,C 180,E1 24653.757,E2 24653.757} C_VEL
LIN {X 0,Y 146.037,Z 369.793,A -85,B 0,C 180,E1 24658.952,E2 24658.952} C_VEL
LIN {X 0,Y 146.067,Z 369.443,A -85,B 0,C 180,E1 24659.518,E2 24659.518} C_VEL
LIN {X 0,Y 146.26,Z 368.263,A -85,B 0,C 180,E1 24662.55,E2 24662.55} C_VEL
LIN {X 0,Y 147.425,Z 375.778,A -85,B 0,C 180,E1 24672.714,E2 24672.714} C_VEL
LIN {X 0,Y 145.413,Z 399.277,A -85,B 0,C 180,E1 24680.934,E2 24680.934} C_VEL
LIN {X 0,Y 143.084,Z 411.307,A -85,B 0,C 180,E1 24684.642,E2 24684.642} C_VEL
LIN {X 0,Y 130.492,Z 434.517,A -85,B 0,C 180,E1 24689.008,E2 24689.008} C_VEL
LIN {X 0,Y 115.915,Z 453.949,A -85,B 0,C 180,E1 24695.97,E2 24695.97} C_VEL
LIN {X 0,Y 101.253,Z 469.368,A -85,B 0,C 180,E1 24706.997,E2 24706.997} C_VEL
LIN {X 0,Y 91.91,Z 478.312,A -85,B 0,C 180,E1 24720.489,E2 24720.489} C_VEL
LIN {X 0,Y 89.113,Z 481.511,A -85,B 0,C 180,E1 24730.201,E2 24730.201} C_VEL
LIN {X 0,Y 88.698,Z 482.949,A -85,B 0,C 180,E1 24740.202,E2 24740.202} C_VEL
LIN {X 0,Y 90.166,Z 482.489,A -85,B 0,C 180,E1 24749.997,E2 24749.997} C_VEL
LIN {X 0,Y 89.427,Z 481.383,A -85,B 0,C 180,E1 24754.837,E2 24754.837} C_VEL
LIN {X 0,Y 89.193,Z 482.09,A -85,B 0,C 180,E1 24769.775,E2 24769.775} C_VEL
LIN {X 0,Y 98.843,Z 478.408,A -85,B 0,C 180,E1 24790.323,E2 24790.323} C_VEL
LIN {X 0,Y 119.726,Z 468.746,A -85,B 0,C 180,E1 24805.819,E2 24805.819} C_VEL
LIN {X 0,Y 144.802,Z 453.78,A -85,B 0,C 180,E1 24815.122,E2 24815.122} C_VEL
LIN {X 0,Y 168.194,Z 435.532,A -85,B 0,C 180,E1 24820.321,E2 24820.321} C_VEL
LIN {X 0,Y 169.549,Z 433.892,A -85,B 0,C 180,E1 24821.283,E2 24821.283} C_VEL
LIN {X 0,Y 169.276,Z 432.679,A -85,B 0,C 180,E1 24824.521,E2 24824.521} C_VEL
LIN {X 0,Y 167.911,Z 432.595,A -85,B 0,C 180,E1 24829.678,E2 24829.678} C_VEL
LIN {X 0,Y 165.247,Z 434.568,A -85,B 0,C 180,E1 24832.16,E2 24832.16} C_VEL
LIN {X 0,Y 159.469,Z 438.769,A -85,B 0,C 180,E1 24834.146,E2 24834.146} C_VEL
LIN {X 0,Y 139.972,Z 450.327,A -85,B 0,C 180,E1 24840.039,E2 24840.039} C_VEL
LIN {X 0,Y 119.213,Z 458.609,A -85,B 0,C 180,E1 24849.657,E2 24849.657} C_VEL
LIN {X 0,Y 109.942,Z 460.765,A -85,B 0,C 180,E1 24856.108,E2 24856.108} C_VEL
LIN {X 0,Y 99.247,Z 461.341,A -85,B 0,C 180,E1 24867.2,E2 24867.2} C_VEL
LIN {X 0,Y 91.311,Z 457.082,A -85,B 0,C 180,E1 24885.861,E2 24885.861} C_VEL
LIN {X 0,Y 92.442,Z 447.816,A -85,B 0,C 180,E1 24903.577,E2 24903.577} C_VEL
LIN {X 0,Y 94.242,Z 444.803,A -85,B 0,C 180,E1 24908.531,E2 24908.531} C_VEL
LIN {X 0,Y 96.982,Z 446.169,A -85,B 0,C 180,E1 24911.872,E2 24911.872} C_VEL
LIN {X 0,Y 92.323,Z 454.202,A -85,B 0,C 180,E1 24925.315,E2 24925.315} C_VEL
LIN {X 0,Y 91.336,Z 458.083,A -85,B 0,C 180,E1 24939.512,E2 24939.512} C_VEL
LIN {X 0,Y 93.476,Z 458.466,A -85,B 0,C 180,E1 24948.839,E2 24948.839} C_VEL
LIN {X 0,Y 100.508,Z 455.696,A -85,B 0,C 180,E1 24961.703,E2 24961.703} C_VEL
LIN {X 0,Y 113.231,Z 447.022,A -85,B 0,C 180,E1 24974.402,E2 24974.402} C_VEL
LIN {X 0,Y 128.047,Z 432.812,A -85,B 0,C 180,E1 24983.598,E2 24983.598} C_VEL
LIN {X 0,Y 141.627,Z 414.809,A -85,B 0,C 180,E1 24989.676,E2 24989.676} C_VEL
LIN {X 0,Y 144.636,Z 409.217,A -85,B 0,C 180,E1 24991.269,E2 24991.269} C_VEL
LIN {X 0,Y 147.263,Z 394.815,A -85,B 0,C 180,E1 24998.074,E2 24998.074} C_VEL
LIN {X 0,Y 147.181,Z 381.855,A -85,B 0,C 180,E1 25005.868,E2 25005.868} C_VEL
LIN {X 0,Y 146.193,Z 372.294,A -85,B 0,C 180,E1 25014.781,E2 25014.781} C_VEL
LIN {X 0,Y 146.067,Z 369.443,A -85,B 0,C 180,E1 25019.518,E2 25019.518} C_VEL
LIN {X 0,Y 145.729,Z 370.676,A -85,B 0,C 180,E1 25022.201,E2 25022.201} C_VEL
LIN {X 0,Y 144.271,Z 379.362,A -85,B 0,C 180,E1 25027.312,E2 25027.312} C_VEL
LIN {X 0,Y 144.329,Z 379.768,A -85,B 0,C 180,E1 25027.916,E2 25027.916} C_VEL
LIN {X 0,Y 144.716,Z 383.681,A -85,B 0,C 180,E1 25031.809,E2 25031.809} C_VEL
LIN {X 0,Y 140.114,Z 409.313,A -85,B 0,C 180,E1 25040.862,E2 25040.862} C_VEL
LIN {X 0,Y 137.818,Z 415.341,A -85,B 0,C 180,E1 25042.284,E2 25042.284} C_VEL
LIN {X 0,Y 123.784,Z 438.103,A -85,B 0,C 180,E1 25046.942,E2 25046.942} C_VEL
LIN {X 0,Y 107.742,Z 456.957,A -85,B 0,C 180,E1 25054.627,E2 25054.627} C_VEL
LIN {X 0,Y 92.623,Z 470.862,A -85,B 0,C 180,E1 25066.534,E2 25066.534} C_VEL
LIN {X 0,Y 82.894,Z 479.058,A -85,B 0,C 180,E1 25082.827,E2 25082.827} C_VEL
LIN {X 0,Y 80.793,Z 481.833,A -85,B 0,C 180,E1 25099.232,E2 25099.232} C_VEL
LIN {X 0,Y 82.227,Z 481.349,A -85,B 0,C 180,E1 25109.997,E2 25109.997} C_VEL
LIN {X 0,Y 81.242,Z 480.247,A -85,B 0,C 180,E1 25118.005,E2 25118.005} C_VEL
LIN {X 0,Y 85.085,Z 479.976,A -85,B 0,C 180,E1 25142.141,E2 25142.141} C_VEL
LIN {X 0,Y 99.252,Z 475.159,A -85,B 0,C 180,E1 25159.477,E2 25159.477} C_VEL
LIN {X 0,Y 123.395,Z 464.344,A -85,B 0,C 180,E1 25172.445,E2 25172.445} C_VEL
LIN {X 0,Y 150.45,Z 447.929,A -85,B 0,C 180,E1 25180.098,E2 25180.098} C_VEL
LIN {X 0,Y 162.334,Z 438.948,A -85,B 0,C 180,E1 25182.336,E2 25182.336} C_VEL
LIN {X 0,Y 163.045,Z 437.779,A -85,B 0,C 180,E1 25183.914,E2 25183.914} C_VEL
LIN {X 0,Y 161.426,Z 437.577,A -85,B 0,C 180,E1 25189.258,E2 25189.258} C_VEL
LIN {X 0,Y 157.334,Z 440.254,A -85,B 0,C 180,E1 25191.412,E2 25191.412} C_VEL
LIN {X 0,Y 135.954,Z 452.179,A -85,B 0,C 180,E1 25197.319,E2 25197.319} C_VEL
LIN {X 0,Y 112.343,Z 460.554,A -85,B 0,C 180,E1 25207.768,E2 25207.768} C_VEL
LIN {X 0,Y 96.449,Z 462.692,A -85,B 0,C 180,E1 25220.168,E2 25220.168} C_VEL
LIN {X 0,Y 84.781,Z 459.628,A -85,B 0,C 180,E1 25239.79,E2 25239.79} C_VEL
LIN {X 0,Y 83.757,Z 450.863,A -85,B 0,C 180,E1 25260.507,E2 25260.507} C_VEL
LIN {X 0,Y 85.736,Z 447.033,A -85,B 0,C 180,E1 25267.49,E2 25267.49} C_VEL
LIN {X 0,Y 88.953,Z 449.018,A -85,B 0,C 180,E1 25272.733,E2 25272.733} C_VEL
LIN {X 0,Y 83.633,Z 457.111,A -85,B 0,C 180,E1 25290.003,E2 25290.003} C_VEL
LIN {X 0,Y 83.59,Z 459.197,A -85,B 0,C 180,E1 25300.403,E2 25300.403} C_VEL
LIN {X 0,Y 86.062,Z 459.536,A -85,B 0,C 180,E1 25310.532,E2 25310.532} C_VEL
LIN {X 0,Y 93.892,Z 456.69,A -85,B 0,C 180,E1 25324.232,E2 25324.232} C_VEL
LIN {X 0,Y 107.741,Z 447.913,A -85,B 0,C 180,E1 25337.336,E2 25337.336} C_VEL
LIN {X 0,Y 123.511,Z 433.573,A -85,B 0,C 180,E1 25346.557,E2 25346.557} C_VEL
LIN {X 0,Y 137.813,Z 415.364,A -85,B 0,C 180,E1 25352.516,E2 25352.516} C_VEL
LIN {X 0,Y 140.605,Z 409.126,A -85,B 0,C 180,E1 25354.964,E2 25354.964} C_VEL
LIN {X 0,Y 143.286,Z 395.846,A -85,B 0,C 180,E1 25361.989,E2 25361.989} C_VEL
LIN {X 0,Y 143.721,Z 385.004,A -85,B 0,C 180,E1 25369.827,E2 25369.827} C_VEL
LIN {X 0,Y 143.781,Z 378.47,A -85,B 0,C 180,E1 25377.707,E2 25377.707} C_VEL
LIN {X 0,Y 144.325,Z 376.203,A -85,B 0,C 180,E1 25382.397,E2 25382.397} C_VEL
LIN {X 0,Y 144.329,Z 379.768,A -85,B 0,C 180,E1 25387.916,E2 25387.916} C_VEL
LIN {X 0,Y 143.882,Z 383.892,A -85,B 0,C 180,E1 25390.121,E2 25390.121} C_VEL
LIN {X 0,Y 139.642,Z 398.733,A -85,B 0,C 180,E1 25393.333,E2 25393.333} C_VEL
LIN {X 0,Y 134.949,Z 414.997,A -85,B 0,C 180,E1 25399.166,E2 25399.166} C_VEL
LIN {X 0,Y 121.145,Z 436.407,A -85,B 0,C 180,E1 25403.267,E2 25403.267} C_VEL
LIN {X 0,Y 104.738,Z 454.762,A -85,B 0,C 180,E1 25410.177,E2 25410.177} C_VEL
LIN {X 0,Y 89.359,Z 468.062,A -85,B 0,C 180,E1 25420.54,E2 25420.54} C_VEL
LIN {X 0,Y 78.18,Z 476.267,A -85,B 0,C 180,E1 25434.612,E2 25434.612} C_VEL
LIN {X 0,Y 74.076,Z 479.368,A -85,B 0,C 180,E1 25445.954,E2 25445.954} C_VEL
LIN {X 0,Y 72.895,Z 480.713,A -85,B 0,C 180,E1 25458.049,E2 25458.049} C_VEL
LIN {X 0,Y 74.288,Z 480.209,A -85,B 0,C 180,E1 25469.997,E2 25469.997} C_VEL
LIN {X 0,Y 73.425,Z 478.784,A -85,B 0,C 180,E1 25478.863,E2 25478.863} C_VEL
LIN {X 0,Y 78.366,Z 478.854,A -85,B 0,C 180,E1 25505.283,E2 25505.283} C_VEL
LIN {X 0,Y 94.19,Z 474.339,A -85,B 0,C 180,E1 25523.225,E2 25523.225} C_VEL
LIN {X 0,Y 119.888,Z 463.996,A -85,B 0,C 180,E1 25535.853,E2 25535.853} C_VEL
LIN {X 0,Y 147.936,Z 448.172,A -85,B 0,C 180,E1 25542.99,E2 25542.99} C_VEL
LIN {X 0,Y 154.863,Z 443.418,A -85,B 0,C 180,E1 25544.195,E2 25544.195} C_VEL
LIN {X 0,Y 156.041,Z 442.31,A -85,B 0,C 180,E1 25545.245,E2 25545.245} C_VEL
LIN {X 0,Y 153.724,Z 442.897,A -85,B 0,C 180,E1 25548.991,E2 25548.991} C_VEL
LIN {X 0,Y 128.896,Z 455.389,A -85,B 0,C 180,E1 25555.52,E2 25555.52} C_VEL
LIN {X 0,Y 106.088,Z 462.26,A -85,B 0,C 180,E1 25565.353,E2 25565.353} C_VEL
LIN {X 0,Y 87.371,Z 463.77,A -85,B 0,C 180,E1 25580.274,E2 25580.274} C_VEL
LIN {X 0,Y 76.275,Z 459.492,A -85,B 0,C 180,E1 25601.787,E2 25601.787} C_VEL
LIN {X 0,Y 76.512,Z 449.953,A -85,B 0,C 180,E1 25623.872,E2 25623.872} C_VEL
LIN {X 0,Y 77.689,Z 449.508,A -85,B 0,C 180,E1 25627.144,E2 25627.144} C_VEL
LIN {X 0,Y 79.951,Z 450.625,A -85,B 0,C 180,E1 25630.892,E2 25630.892} C_VEL
LIN {X 0,Y 79.69,Z 452.546,A -85,B 0,C 180,E1 25634.998,E2 25634.998} C_VEL
LIN {X 0,Y 75.607,Z 458.817,A -85,B 0,C 180,E1 25652.285,E2 25652.285} C_VEL
LIN {X 0,Y 78.745,Z 460.598,A -85,B 0,C 180,E1 25672.539,E2 25672.539} C_VEL
LIN {X 0,Y 87.494,Z 457.676,A -85,B 0,C 180,E1 25687.135,E2 25687.135} C_VEL
LIN {X 0,Y 102.557,Z 448.802,A -85,B 0,C 180,E1 25700.58,E2 25700.58} C_VEL
LIN {X 0,Y 119.09,Z 434.584,A -85,B 0,C 180,E1 25709.607,E2 25709.607} C_VEL
LIN {X 0,Y 134.353,Z 415.934,A -85,B 0,C 180,E1 25715.503,E2 25715.503} C_VEL
LIN {X 0,Y 138.317,Z 404.301,A -85,B 0,C 180,E1 25721.68,E2 25721.68} C_VEL
LIN {X 0,Y 140.298,Z 392.802,A -85,B 0,C 180,E1 25729.808,E2 25729.808} C_VEL
LIN {X 0,Y 141.059,Z 386.568,A -85,B 0,C 180,E1 25736.785,E2 25736.785} C_VEL
LIN {X 0,Y 141.864,Z 383.809,A -85,B 0,C 180,E1 25741.569,E2 25741.569} C_VEL
LIN {X 0,Y 141.815,Z 389.502,A -85,B 0,C 180,E1 25749.919,E2 25749.919} C_VEL
LIN {X 0,Y 139.642,Z 398.733,A -85,B 0,C 180,E1 25753.333,E2 25753.333} C_VEL
LIN {X 0,Y 137.039,Z 406.075,A -85,B 0,C 180,E1 25755.035,E2 25755.035} C_VEL
LIN {X 0,Y 129.965,Z 419.018,A -85,B 0,C 180,E1 25756.531,E2 25756.531} C_VEL
LIN {X 0,Y 114.939,Z 439.63,A -85,B 0,C 180,E1 25760.699,E2 25760.699} C_VEL
LIN {X 0,Y 96.508,Z 457.788,A -85,B 0,C 180,E1 25768.411,E2 25768.411} C_VEL
LIN {X 0,Y 79.544,Z 470.302,A -85,B 0,C 180,E1 25780.635,E2 25780.635} C_VEL
LIN {X 0,Y 68.794,Z 476.97,A -85,B 0,C 180,E1 25796.74,E2 25796.74} C_VEL
LIN {X 0,Y 65.044,Z 479.593,A -85,B 0,C 180,E1 25816.581,E2 25816.581} C_VEL
LIN {X 0,Y 66.329,Z 479.066,A -85,B 0,C 180,E1 25829.996,E2 25829.996} C_VEL
LIN {X 0,Y 65.598,Z 477.295,A -85,B 0,C 180,E1 25839.931,E2 25839.931} C_VEL
LIN {X 0,Y 71.904,Z 477.705,A -85,B 0,C 180,E1 25869.015,E2 25869.015} C_VEL
LIN {X 0,Y 94.721,Z 472.012,A -85,B 0,C 180,E1 25890.432,E2 25890.432} C_VEL
LIN {X 0,Y 123.449,Z 460.665,A -85,B 0,C 180,E1 25901.315,E2 25901.315} C_VEL
LIN {X 0,Y 147.088,Z 447.646,A -85,B 0,C 180,E1 25906.183,E2 25906.183} C_VEL
LIN {X 0,Y 147.614,Z 447.118,A -85,B 0,C 180,E1 25907.01,E2 25907.01} C_VEL
LIN {X 0,Y 121.458,Z 458.589,A -85,B 0,C 180,E1 25913.66,E2 25913.66} C_VEL
LIN {X 0,Y 105.183,Z 463.019,A -85,B 0,C 180,E1 25920.051,E2 25920.051} C_VEL
LIN {X 0,Y 89.047,Z 465.095,A -85,B 0,C 180,E1 25929.818,E2 25929.818} C_VEL
LIN {X 0,Y 76.028,Z 464.175,A -85,B 0,C 180,E1 25943.466,E2 25943.466} C_VEL
LIN {X 0,Y 67.396,Z 457.939,A -85,B 0,C 180,E1 25967.806,E2 25967.806} C_VEL
LIN {X 0,Y 68.489,Z 451.153,A -85,B 0,C 180,E1 25983.858,E2 25983.858} C_VEL
LIN {X 0,Y 71.039,Z 452.553,A -85,B 0,C 180,E1 25989.455,E2 25989.455} C_VEL
LIN {X 0,Y 71.959,Z 453.988,A -85,B 0,C 180,E1 25993.856,E2 25993.856} C_VEL
LIN {X 0,Y 67.924,Z 459.451,A -85,B 0,C 180,E1 26010.004,E2 26010.004} C_VEL
LIN {X 0,Y 68.184,Z 461.422,A -85,B 0,C 180,E1 26022.79,E2 26022.79} C_VEL
LIN {X 0,Y 71.536,Z 461.656,A -85,B 0,C 180,E1 26034.957,E2 26034.957} C_VEL
LIN {X 0,Y 81.34,Z 458.659,A -85,B 0,C 180,E1 26050.493,E2 26050.493} C_VEL
LIN {X 0,Y 97.733,Z 449.688,A -85,B 0,C 180,E1 26064.159,E2 26064.159} C_VEL
LIN {X 0,Y 114.518,Z 436.078,A -85,B 0,C 180,E1 26072.684,E2 26072.684} C_VEL
LIN {X 0,Y 129.982,Z 418.326,A -85,B 0,C 180,E1 26078.244,E2 26078.244} C_VEL
LIN {X 0,Y 134.463,Z 407.21,A -85,B 0,C 180,E1 26084.754,E2 26084.754} C_VEL
LIN {X 0,Y 136.944,Z 397.549,A -85,B 0,C 180,E1 26092.633,E2 26092.633} C_VEL
LIN {X 0,Y 138.479,Z 392.368,A -85,B 0,C 180,E1 26099.961,E2 26099.961} C_VEL
LIN {X 0,Y 138.789,Z 392.279,A -85,B 0,C 180,E1 26103.247,E2 26103.247} C_VEL
LIN {X 0,Y 138.742,Z 395.09,A -85,B 0,C 180,E1 26107.93,E2 26107.93} C_VEL
LIN {X 0,Y 131.768,Z 415.715,A -85,B 0,C 180,E1 26115.873,E2 26115.873} C_VEL
LIN {X 0,Y 129.965,Z 419.018,A -85,B 0,C 180,E1 26116.531,E2 26116.531} C_VEL
LIN {X 0,Y 122.476,Z 428.271,A -85,B 0,C 180,E1 26116.365,E2 26116.365} C_VEL
LIN {X 0,Y 115.207,Z 435.721,A -85,B 0,C 180,E1 26116.113,E2 26116.113} C_VEL
LIN {X 0,Y 114.261,Z 436.758,A -85,B 0,C 180,E1 26116.321,E2 26116.321} C_VEL
LIN {X 0,Y 95.503,Z 454.857,A -85,B 0,C 180,E1 26122.819,E2 26122.819} C_VEL
LIN {X 0,Y 77.073,Z 467.815,A -85,B 0,C 180,E1 26133.679,E2 26133.679} C_VEL
LIN {X 0,Y 62.181,Z 475.918,A -85,B 0,C 180,E1 26152.644,E2 26152.644} C_VEL
LIN {X 0,Y 57.224,Z 478.471,A -85,B 0,C 180,E1 26174.706,E2 26174.706} C_VEL
LIN {X 0,Y 58.387,Z 477.924,A -85,B 0,C 180,E1 26189.996,E2 26189.996} C_VEL
LIN {X 0,Y 57.778,Z 475.738,A -85,B 0,C 180,E1 26201.292,E2 26201.292} C_VEL
LIN {X 0,Y 65.828,Z 476.478,A -85,B 0,C 180,E1 26233.443,E2 26233.443} C_VEL
LIN {X 0,Y 90.517,Z 471.408,A -85,B 0,C 180,E1 26254.624,E2 26254.624} C_VEL
LIN {X 0,Y 121.122,Z 460.5,A -85,B 0,C 180,E1 26264.905,E2 26264.905} C_VEL
LIN {X 0,Y 128.778,Z 456.961,A -85,B 0,C 180,E1 26266.489,E2 26266.489} C_VEL
LIN {X 0,Y 129.391,Z 456.47,A -85,B 0,C 180,E1 26267.402,E2 26267.402} C_VEL
LIN {X 0,Y 106.145,Z 463.496,A -85,B 0,C 180,E1 26274.326,E2 26274.326} C_VEL
LIN {X 0,Y 90.572,Z 465.957,A -85,B 0,C 180,E1 26281.633,E2 26281.633} C_VEL
LIN {X 0,Y 76.996,Z 466.191,A -85,B 0,C 180,E1 26291.518,E2 26291.518} C_VEL
LIN {X 0,Y 62.127,Z 462.125,A -85,B 0,C 180,E1 26314.633,E2 26314.633} C_VEL
LIN {X 0,Y 60.436,Z 453.598,A -85,B 0,C 180,E1 26343.072,E2 26343.072} C_VEL
LIN {X 0,Y 63.751,Z 455.27,A -85,B 0,C 180,E1 26351.497,E2 26351.497} C_VEL
LIN {X 0,Y 60.076,Z 460.615,A -85,B 0,C 180,E1 26370.004,E2 26370.004} C_VEL
LIN {X 0,Y 60.537,Z 462.536,A -85,B 0,C 180,E1 26384.438,E2 26384.438} C_VEL
LIN {X 0,Y 64.511,Z 462.709,A -85,B 0,C 180,E1 26397.897,E2 26397.897} C_VEL
LIN {X 0,Y 77.565,Z 458.823,A -85,B 0,C 180,E1 26416.485,E2 26416.485} C_VEL
LIN {X 0,Y 93.321,Z 450.567,A -85,B 0,C 180,E1 26428.1,E2 26428.1} C_VEL
LIN {X 0,Y 112.444,Z 435.619,A -85,B 0,C 180,E1 26436.785,E2 26436.785} C_VEL
LIN {X 0,Y 126.243,Z 420.087,A -85,B 0,C 180,E1 26441.555,E2 26441.555} C_VEL
LIN {X 0,Y 130.947,Z 409.905,A -85,B 0,C 180,E1 26448.323,E2 26448.323} C_VEL
LIN {X 0,Y 133.591,Z 402.815,A -85,B 0,C 180,E1 26455.041,E2 26455.041} C_VEL
LIN {X 0,Y 134.984,Z 399.725,A -85,B 0,C 180,E1 26459.96,E2 26459.96} C_VEL
LIN {X 0,Y 135.268,Z 400.493,A -85,B 0,C 180,E1 26464.847,E2 26464.847} C_VEL
LIN {X 0,Y 134.595,Z 402.865,A -85,B 0,C 180,E1 26466.785,E2 26466.785} C_VEL
LIN {X 0,Y 127.123,Z 419.796,A -85,B 0,C 180,E1 26473.273,E2 26473.273} C_VEL
LIN {X 0,Y 114.261,Z 436.758,A -85,B 0,C 180,E1 26476.321,E2 26476.321} C_VEL
LIN {X 0,Y 101.328,Z 448.297,A -85,B 0,C 180,E1 26477.881,E2 26477.881} C_VEL
LIN {X 0,Y 88.966,Z 456.812,A -85,B 0,C 180,E1 26479.774,E2 26479.774} C_VEL
LIN {X 0,Y 87.345,Z 457.909,A -85,B 0,C 180,E1 26480.393,E2 26480.393} C_VEL
LIN {X 0,Y 67.871,Z 469.486,A -85,B 0,C 180,E1 26492.33,E2 26492.33} C_VEL
LIN {X 0,Y 52.775,Z 476.147,A -85,B 0,C 180,E1 26515.114,E2 26515.114} C_VEL
LIN {X 0,Y 49.494,Z 477.349,A -85,B 0,C 180,E1 26532.244,E2 26532.244} C_VEL
LIN {X 0,Y 50.432,Z 476.775,A -85,B 0,C 180,E1 26549.995,E2 26549.995} C_VEL
LIN {X 0,Y 50.075,Z 474.533,A -85,B 0,C 180,E1 26567.533,E2 26567.533} C_VEL
LIN {X 0,Y 60.215,Z 475.252,A -85,B 0,C 180,E1 26598.74,E2 26598.74} C_VEL
LIN {X 0,Y 82.011,Z 471.874,A -85,B 0,C 180,E1 26616.918,E2 26616.918} C_VEL
LIN {X 0,Y 108.696,Z 464.313,A -85,B 0,C 180,E1 26626.349,E2 26626.349} C_VEL
LIN {X 0,Y 111.504,Z 463.094,A -85,B 0,C 180,E1 26627.849,E2 26627.849} C_VEL
LIN {X 0,Y 90.859,Z 466.866,A -85,B 0,C 180,E1 26635.162,E2 26635.162} C_VEL
LIN {X 0,Y 75.625,Z 467.569,A -85,B 0,C 180,E1 26643.952,E2 26643.952} C_VEL
LIN {X 0,Y 56.987,Z 464.197,A -85,B 0,C 180,E1 26666.341,E2 26666.341} C_VEL
LIN {X 0,Y 52.1,Z 455.664,A -85,B 0,C 180,E1 26700.544,E2 26700.544} C_VEL
LIN {X 0,Y 54.464,Z 456.82,A -85,B 0,C 180,E1 26708.194,E2 26708.194} C_VEL
LIN {X 0,Y 55.347,Z 458.056,A -85,B 0,C 180,E1 26714.183,E2 26714.183} C_VEL
LIN {X 0,Y 52.22,Z 461.774,A -85,B 0,C 180,E1 26730.005,E2 26730.005} C_VEL
LIN {X 0,Y 52.958,Z 463.648,A -85,B 0,C 180,E1 26746.56,E2 26746.56} C_VEL
LIN {X 0,Y 57.669,Z 463.767,A -85,B 0,C 180,E1 26761.561,E2 26761.561} C_VEL
LIN {X 0,Y 72.981,Z 459.565,A -85,B 0,C 180,E1 26781.567,E2 26781.567} C_VEL
LIN {X 0,Y 92.443,Z 449.569,A -85,B 0,C 180,E1 26793.875,E2 26793.875} C_VEL
LIN {X 0,Y 111.569,Z 434.476,A -85,B 0,C 180,E1 26801.228,E2 26801.228} C_VEL
LIN {X 0,Y 122.503,Z 422.438,A -85,B 0,C 180,E1 26804.78,E2 26804.78} C_VEL
LIN {X 0,Y 127.36,Z 413.719,A -85,B 0,C 180,E1 26811.303,E2 26811.303} C_VEL
LIN {X 0,Y 129.834,Z 408.829,A -85,B 0,C 180,E1 26816.627,E2 26816.627} C_VEL
LIN {X 0,Y 131.049,Z 406.905,A -85,B 0,C 180,E1 26819.959,E2 26819.959} C_VEL
LIN {X 0,Y 131.442,Z 407.213,A -85,B 0,C 180,E1 26824.074,E2 26824.074} C_VEL
LIN {X 0,Y 124.546,Z 420.719,A -85,B 0,C 180,E1 26829.871,E2 26829.871} C_VEL
LIN {X 0,Y 106.809,Z 441.769,A -85,B 0,C 180,E1 26833.752,E2 26833.752} C_VEL
LIN {X 0,Y 87.345,Z 457.909,A -85,B 0,C 180,E1 26840.393,E2 26840.393} C_VEL
LIN {X 0,Y 72.6,Z 465.556,A -85,B 0,C 180,E1 26844.515,E2 26844.515} C_VEL
LIN {X 0,Y 59.458,Z 470.429,A -85,B 0,C 180,E1 26850.019,E2 26850.019} C_VEL
LIN {X 0,Y 57.898,Z 471.005,A -85,B 0,C 180,E1 26851.413,E2 26851.413} C_VEL
LIN {X 0,Y 46.35,Z 475.074,A -85,B 0,C 180,E1 26869.366,E2 26869.366} C_VEL
LIN {X 0,Y 41.877,Z 476.226,A -85,B 0,C 180,E1 26888.873,E2 26888.873} C_VEL
LIN {X 0,Y 42.475,Z 475.619,A -85,B 0,C 180,E1 26909.994,E2 26909.994} C_VEL
LIN {X 0,Y 42.554,Z 472.901,A -85,B 0,C 180,E1 26930.763,E2 26930.763} C_VEL
LIN {X 0,Y 59.399,Z 473.709,A -85,B 0,C 180,E1 26969.568,E2 26969.568} C_VEL
LIN {X 0,Y 87.321,Z 469.318,A -85,B 0,C 180,E1 26985.399,E2 26985.399} C_VEL
LIN {X 0,Y 94.216,Z 467.507,A -85,B 0,C 180,E1 26988.198,E2 26988.198} C_VEL
LIN {X 0,Y 69.391,Z 468.645,A -85,B 0,C 180,E1 27000.078,E2 27000.078} C_VEL
LIN {X 0,Y 49.439,Z 464.671,A -85,B 0,C 180,E1 27023.71,E2 27023.71} C_VEL
LIN {X 0,Y 43.689,Z 457.431,A -85,B 0,C 180,E1 27055.138,E2 27055.138} C_VEL
LIN {X 0,Y 47.153,Z 459.374,A -85,B 0,C 180,E1 27071.341,E2 27071.341} C_VEL
LIN {X 0,Y 44.365,Z 462.926,A -85,B 0,C 180,E1 27090.006,E2 27090.006} C_VEL
LIN {X 0,Y 45.491,Z 464.759,A -85,B 0,C 180,E1 27109.379,E2 27109.379} C_VEL
LIN {X 0,Y 51.143,Z 464.821,A -85,B 0,C 180,E1 27126.171,E2 27126.171} C_VEL
LIN {X 0,Y 66.706,Z 461.102,A -85,B 0,C 180,E1 27145.426,E2 27145.426} C_VEL
LIN {X 0,Y 86.019,Z 452.315,A -85,B 0,C 180,E1 27157.078,E2 27157.078} C_VEL
LIN {X 0,Y 106.428,Z 437.786,A -85,B 0,C 180,E1 27164.357,E2 27164.357} C_VEL
LIN {X 0,Y 118.502,Z 425.635,A -85,B 0,C 180,E1 27167.723,E2 27167.723} C_VEL
LIN {X 0,Y 123.757,Z 417.85,A -85,B 0,C 180,E1 27174.306,E2 27174.306} C_VEL
LIN {X 0,Y 126.577,Z 413.883,A -85,B 0,C 180,E1 27179.957,E2 27179.957} C_VEL
LIN {X 0,Y 127.022,Z 413.517,A -85,B 0,C 180,E1 27181.524,E2 27181.524} C_VEL
LIN {X 0,Y 125.75,Z 415.911,A -85,B 0,C 180,E1 27183.559,E2 27183.559} C_VEL
LIN {X 0,Y 120.647,Z 423.979,A -85,B 0,C 180,E1 27186.71,E2 27186.71} C_VEL
LIN {X 0,Y 101.61,Z 444.277,A -85,B 0,C 180,E1 27190.292,E2 27190.292} C_VEL
LIN {X 0,Y 79.131,Z 460.626,A -85,B 0,C 180,E1 27197.534,E2 27197.534} C_VEL
LIN {X 0,Y 57.898,Z 471.005,A -85,B 0,C 180,E1 27211.413,E2 27211.413} C_VEL
LIN {X 0,Y 44.479,Z 474.341,A -85,B 0,C 180,E1 27223.621,E2 27223.621} C_VEL
LIN {X 0,Y 34.373,Z 475.084,A -85,B 0,C 180,E1 27244.735,E2 27244.735} C_VEL
LIN {X 0,Y 34.496,Z 474.455,A -85,B 0,C 180,E1 27269.993,E2 27269.993} C_VEL
LIN {X 0,Y 35.24,Z 471.233,A -85,B 0,C 180,E1 27295.346,E2 27295.346} C_VEL
LIN {X 0,Y 51.047,Z 472.668,A -85,B 0,C 180,E1 27332.466,E2 27332.466} C_VEL
LIN {X 0,Y 76.956,Z 470.032,A -85,B 0,C 180,E1 27348.63,E2 27348.63} C_VEL
LIN {X 0,Y 51.304,Z 467.995,A -85,B 0,C 180,E1 27365.716,E2 27365.716} C_VEL
LIN {X 0,Y 36.377,Z 460.794,A -85,B 0,C 180,E1 27401.192,E2 27401.192} C_VEL
LIN {X 0,Y 35.796,Z 459.448,A -85,B 0,C 180,E1 27409.66,E2 27409.66} C_VEL
LIN {X 0,Y 38.704,Z 461.605,A -85,B 0,C 180,E1 27433.004,E2 27433.004} C_VEL
LIN {X 0,Y 38.161,Z 465.872,A -85,B 0,C 180,E1 27473.3,E2 27473.3} C_VEL
LIN {X 0,Y 45.025,Z 465.879,A -85,B 0,C 180,E1 27492.097,E2 27492.097} C_VEL
LIN {X 0,Y 60.964,Z 462.565,A -85,B 0,C 180,E1 27510.224,E2 27510.224} C_VEL
LIN {X 0,Y 83.259,Z 453.188,A -85,B 0,C 180,E1 27522.095,E2 27522.095} C_VEL
LIN {X 0,Y 105.066,Z 438.091,A -85,B 0,C 180,E1 27528.647,E2 27528.647} C_VEL
LIN {X 0,Y 114.241,Z 429.368,A -85,B 0,C 180,E1 27530.715,E2 27530.715} C_VEL
LIN {X 0,Y 119.529,Z 423.007,A -85,B 0,C 180,E1 27536.339,E2 27536.339} C_VEL
LIN {X 0,Y 122.132,Z 420.158,A -85,B 0,C 180,E1 27540.854,E2 27540.854} C_VEL
LIN {X 0,Y 118.427,Z 425.293,A -85,B 0,C 180,E1 27543.106,E2 27543.106} C_VEL
LIN {X 0,Y 98.652,Z 445.012,A -85,B 0,C 180,E1 27546.123,E2 27546.123} C_VEL
LIN {X 0,Y 77.078,Z 459.723,A -85,B 0,C 180,E1 27551.782,E2 27551.782} C_VEL
LIN {X 0,Y 54.388,Z 469.893,A -85,B 0,C 180,E1 27563.799,E2 27563.799} C_VEL
LIN {X 0,Y 40.544,Z 473.998,A -85,B 0,C 180,E1 27581.885,E2 27581.885} C_VEL
LIN {X 0,Y 34.373,Z 475.084,A -85,B 0,C 180,E1 27604.735,E2 27604.735} C_VEL
LIN {X 0,Y 31.012,Z 474.546,A -85,B 0,C 180,E1 27618.824,E2 27618.824} C_VEL
LIN {X 0,Y 26.552,Z 471.701,A -85,B 0,C 180,E1 27647.673,E2 27647.673} C_VEL
LIN {X 0,Y 29.401,Z 469.873,A -85,B 0,C 180,E1 27668.428,E2 27668.428} C_VEL
LIN {X 0,Y 54.83,Z 471.154,A -85,B 0,C 180,E1 27705.775,E2 27705.775} C_VEL
LIN {X 0,Y 59.671,Z 470.727,A -85,B 0,C 180,E1 27709.15,E2 27709.15} C_VEL
LIN {X 0,Y 35.38,Z 465.672,A -85,B 0,C 180,E1 27733.852,E2 27733.852} C_VEL
LIN {X 0,Y 28.421,Z 461.399,A -85,B 0,C 180,E1 27760.921,E2 27760.921} C_VEL
LIN {X 0,Y 28.862,Z 462.46,A -85,B 0,C 180,E1 27778.488,E2 27778.488} C_VEL
LIN {X 0,Y 30.234,Z 463.693,A -85,B 0,C 180,E1 27795.557,E2 27795.557} C_VEL
LIN {X 0,Y 31.091,Z 466.985,A -85,B 0,C 180,E1 27839.044,E2 27839.044} C_VEL
LIN {X 0,Y 39.535,Z 466.937,A -85,B 0,C 180,E1 27859.772,E2 27859.772} C_VEL
LIN {X 0,Y 60.678,Z 462.605,A -85,B 0,C 180,E1 27878.978,E2 27878.978} C_VEL
LIN {X 0,Y 81.178,Z 454.062,A -85,B 0,C 180,E1 27887.412,E2 27887.412} C_VEL
LIN {X 0,Y 102.689,Z 439.767,A -85,B 0,C 180,E1 27892.704,E2 27892.704} C_VEL
LIN {X 0,Y 111.178,Z 432.112,A -85,B 0,C 180,E1 27894.308,E2 27894.308} C_VEL
LIN {X 0,Y 115.574,Z 427.722,A -85,B 0,C 180,E1 27898.985,E2 27898.985} C_VEL
LIN {X 0,Y 110.488,Z 433.182,A -85,B 0,C 180,E1 27899.951,E2 27899.951} C_VEL
LIN {X 0,Y 88.772,Z 451.042,A -85,B 0,C 180,E1 27902.904,E2 27902.904} C_VEL
LIN {X 0,Y 64.953,Z 463.981,A -85,B 0,C 180,E1 27909.092,E2 27909.092} C_VEL
LIN {X 0,Y 41.352,Z 471.701,A -85,B 0,C 180,E1 27924.161,E2 27924.161} C_VEL
LIN {X 0,Y 26.753,Z 473.879,A -85,B 0,C 180,E1 27961.166,E2 27961.166} C_VEL
LIN {X 0,Y 26.511,Z 473.288,A -85,B 0,C 180,E1 27989.991,E2 27989.991} C_VEL
LIN {X 0,Y 26.552,Z 471.701,A -85,B 0,C 180,E1 28007.673,E2 28007.673} C_VEL
LIN {X 0,Y 28.156,Z 469.786,A -85,B 0,C 180,E1 28034.76,E2 28034.76} C_VEL
LIN {X 0,Y 39.96,Z 469.657,A -85,B 0,C 180,E1 28067.169,E2 28067.169} C_VEL
LIN {X 0,Y 42.845,Z 469.771,A -85,B 0,C 180,E1 28069.446,E2 28069.446} C_VEL
LIN {X 0,Y 22.406,Z 463.215,A -85,B 0,C 180,E1 28105.463,E2 28105.463} C_VEL
LIN {X 0,Y 21.772,Z 465.099,A -85,B 0,C 180,E1 28151.051,E2 28151.051} C_VEL
LIN {X 0,Y 24.514,Z 468.094,A -85,B 0,C 180,E1 28208.006,E2 28208.006} C_VEL
LIN {X 0,Y 34.969,Z 467.994,A -85,B 0,C 180,E1 28229.674,E2 28229.674} C_VEL
LIN {X 0,Y 55.257,Z 464.427,A -85,B 0,C 180,E1 28244.852,E2 28244.852} C_VEL
LIN {X 0,Y 79.83,Z 454.936,A -85,B 0,C 180,E1 28252.952,E2 28252.952} C_VEL
LIN {X 0,Y 98.499,Z 443.225,A -85,B 0,C 180,E1 28256.562,E2 28256.562} C_VEL
LIN {X 0,Y 73.75,Z 458.721,A -85,B 0,C 180,E1 28259.927,E2 28259.927} C_VEL
LIN {X 0,Y 49.396,Z 468.071,A -85,B 0,C 180,E1 28266.823,E2 28266.823} C_VEL
LIN {X 0,Y 32.061,Z 471.821,A -85,B 0,C 180,E1 28279.702,E2 28279.702} C_VEL
LIN {X 0,Y 20.861,Z 472.868,A -85,B 0,C 180,E1 28305.962,E2 28305.962} C_VEL
LIN {X 0,Y 18.51,Z 472.119,A -85,B 0,C 180,E1 28349.987,E2 28349.987} C_VEL
LIN {X 0,Y 23.889,Z 468.213,A -85,B 0,C 180,E1 28401.115,E2 28401.115} C_VEL
LIN {X 0,Y 39.96,Z 469.657,A -85,B 0,C 180,E1 28427.169,E2 28427.169} C_VEL
LIN {X 0,Y 38.125,Z 468.912,A -85,B 0,C 180,E1 28432.176,E2 28432.176} C_VEL
LIN {X 0,Y 31.583,Z 467.732,A -85,B 0,C 180,E1 28437.572,E2 28437.572} C_VEL
LIN {X 0,Y 13.751,Z 466.085,A -85,B 0,C 180,E1 28471.965,E2 28471.965} C_VEL
LIN {X 0,Y 12.97,Z 466.267,A -85,B 0,C 180,E1 28484.742,E2 28484.742} C_VEL
LIN {X 0,Y 13.125,Z 466.565,A -85,B 0,C 180,E1 28499.773,E2 28499.773} C_VEL
LIN {X 0,Y 12.979,Z 467.518,A -85,B 0,C 180,E1 28530.019,E2 28530.019} C_VEL
LIN {X 0,Y 18.944,Z 469.197,A -85,B 0,C 180,E1 28582.823,E2 28582.823} C_VEL
LIN {X 0,Y 31.729,Z 469.053,A -85,B 0,C 180,E1 28602.045,E2 28602.045} C_VEL
LIN {X 0,Y 56.911,Z 464.542,A -85,B 0,C 180,E1 28613.931,E2 28613.931} C_VEL
LIN {X 0,Y 60.575,Z 463.488,A -85,B 0,C 180,E1 28615.217,E2 28615.217} C_VEL
LIN {X 0,Y 40.685,Z 469.004,A -85,B 0,C 180,E1 28619.867,E2 28619.867} C_VEL
LIN {X 0,Y 16.531,Z 471.73,A -85,B 0,C 180,E1 28644.066,E2 28644.066} C_VEL
LIN {X 0,Y 10.489,Z 470.947,A -85,B 0,C 180,E1 28709.977,E2 28709.977} C_VEL
LIN {X 0,Y 19.898,Z 466.396,A -85,B 0,C 180,E1 28779.147,E2 28779.147} C_VEL
LIN {X 0,Y 24.361,Z 467.038,A -85,B 0,C 180,E1 28786.745,E2 28786.745} C_VEL
LIN {X 0,Y 21.927,Z 465.815,A -85,B 0,C 180,E1 28795.395,E2 28795.395} C_VEL
LIN {X 0,Y 19.541,Z 464.921,A -85,B 0,C 180,E1 28800.276,E2 28800.276} C_VEL
LIN {X 0,Y 12.97,Z 466.267,A -85,B 0,C 180,E1 28844.742,E2 28844.742} C_VEL
LIN {X 0,Y 10.416,Z 467.533,A -85,B 0,C 180,E1 28875.415,E2 28875.415} C_VEL
LIN {X 0,Y 14.02,Z 470.126,A -85,B 0,C 180,E1 28964.581,E2 28964.581} C_VEL
LIN {X 0,Y 19.234,Z 470.511,A -85,B 0,C 180,E1 28972.649,E2 28972.649} C_VEL
LIN {X 0,Y 2.47,Z 469.775,A -85,B 0,C 180,E1 29069.9,E2 29069.9} C_VEL
LIN {X 0,Y 8.119,Z 467.936,A -85,B 0,C 180,E1 29160.664,E2 29160.664} C_VEL
LIN {X 0,Y 4.987,Z 468.685,A -85,B 0,C 180,E1 29250.049,E2 29250.049} C_VEL
LIN {X 0,Y 14.02,Z 470.126,A -85,B 0,C 180,E1 29324.581,E2 29324.581} C_VEL
LIN {X 0,Y 15.706,Z 472.114,A -85,B 0,C 180,E1 29326.893,E2 29326.893} C_VEL
LIN {X 0,Y 15.706,Z 550,A -85,B 0,C 180,E1 29326.893,E2 29326.893} C_VEL
LIN {X 0,Y 15.706,Z 550,A -85,B 0,C 180,E1 29326.893,E2 29326.893}

